TYPE EL6001_Data :
STRUCT
	{attribute addProperty Name "COM Inputs"}
	COM_Inputs : EL6001_COM_Inputs;
	{attribute addProperty Name "COM Outputs"}
	COM_Outputs : EL6001_COM_Outputs;
END_STRUCT
END_TYPE

(* stored: Version 1.1.0.1, ProductVersion 3.1.4024.9
   DUT EL6001_Data: Id {ba49c726-a0bb-0090-179c-8c191d46b9ec} *)
